TYPE ST_ReferenceBindingFileConfig :
STRUCT
	Source : STRING(255);
	TargetPort : STRING(80);
END_STRUCT
END_TYPE

(* stored: Version 1.1.0.1, ProductVersion 3.1.4026.18
   DUT ST_ReferenceBindingFileConfig: Id {2ba99eb3-f07e-48cb-82b0-27bc4b65be4d} *)
